{attribute addProperty BoxType ""}
{attribute addProperty Id "_defaultSyncUnitTasks_486549DC19524.3750A_0013_EL9221_4030_0018SyncUnitTasks_486549DC19524.3750A_0014_EL9221_5000_0018SyncUnitTasks_486549DC19524.3750A_0015_EL9221_5090_0018SyncUnitTasks_486549DC19524.3750A_0016_EL9221_6000_0018SyncUnitTasks_486549DC19524.3750A_0017_EL9221_6040_0018SyncUnitTasks_486549DC19524.3750A_0018_EL9221_9060_0018SyncUnitTasks_486549DC19524.3750A_0019_EL9221_9080_0018SyncUnitTasks_486549DC19524.3750A_0020_EL9222_4433_0018SyncUnitTasks_486549DC19524.3750A_0021_EL9222_5500_0018SyncUnitTasks_486549DC19524.3750A_0022_EL9222_6600_0018SyncUnitTasks_486549DC19524.3750A_0023_EL9222_6644_0018SyncUnitTasks_486549DC19524.3750A_0024_EL9222_9482_0018SyncUnitTasks_486549DC19524.3750A_0025_EL9222_9664_0018SyncUnitTasks_486549DC19524.3750A_0026_EL9227_4433_0018SyncUnitTasks_486549DC19524.3750A_0027_EL9227_5500_0018SyncUnitTasks_486549DC19524.3750A_0028_EL9227_6600_0018SyncUnitTasks_486549DC19524.3750A_0029_EL9227_6644_0018SyncUnitTasks_486549DC19524.3750A_0030_EL9227_9482_0018SyncUnitTasks_486549DC19524.3750A_0031_EL9227_9664_0018SyncUnitTasks_486549DC19524.3750A_0033_EL6690_0002_0016SyncUnitTasks_486549DC19524.3750A_0034_EL6690_0002_0017SyncUnitTasks_486549DC19524.3750A_0035_EL6690_0002_0018SyncUnitTasks_486549DC19524.3750A_0036_EL6690_0002_0019SyncUnitTasks_486549DC19524.3750A_0001_EL6720_0000_0016_0SyncUnitTasks_486549DC19524.3750A_0001_EL6720_0000_0016_1SyncUnitTasks_486549DC19524.3750A_0001_EL6720_0000_0016_2SyncUnitTasks_486549DC19524.3750A_0002_EL6720_0000_0017_0SyncUnitTasks_486549DC19524.3750A_0002_EL6720_0000_0017_1SyncUnitTasks_486549DC19524.3750A_0002_EL6720_0000_0017_2SyncUnitTasks_486549DC19524.3750A_0003_EL6720_0000_0018_0SyncUnitTasks_486549DC19524.3750A_0003_EL6720_0000_0018_1SyncUnitTasks_486549DC19524.3750A_0003_EL6720_0000_0018_2SyncUnitTasks_486549DC19524.3750A_0004_EL6720_0000_0020_0SyncUnitTasks_486549DC19524.3750A_0004_EL6720_0000_0020_1SyncUnitTasks_486549DC19524.3750A_0004_EL6720_0000_0020_2SyncUnitTasks_486549DC19524.3750A_0005_EL6731_0000_0000SyncUnitTasks_486549DC19524.3750A_0006_EL6731_0001_0000SyncUnitTasks_486549DC19524.3750A_0008_EL6731_0000_0017SyncUnitTasks_486549DC19524.3750A_0009_EL6731_0000_0018SyncUnitTasks_486549DC19524.3750A_0010_EL6731_0000_0019SyncUnitTasks_486549DC19524.3750A_0011_EL6731_0000_0020SyncUnitTasks_486549DC19524.3750A_0012_EL6731_0000_0021SyncUnitTasks_486549DC19524.3750A_0013_EL6731_0000_0022SyncUnitTasks_486549DC19524.3750A_0014_EL6731_0000_0023SyncUnitTasks_486549DC19524.3750A_0015_EL6731_0000_0025SyncUnitTasks_486549DC19524.3750A_0016_EL6731_0100_0017SyncUnitTasks_486549DC19524.3750A_0017_EL6731_0100_0018SyncUnitTasks_486549DC19524.3750A_0018_EL6731_0100_0019SyncUnitTasks_486549DC19524.3750A_0020_EL6731_0100_0021SyncUnitTasks_486549DC19524.3750A_0021_EL6731_0100_0022SyncUnitTasks_486549DC19524.3750A_0022_EL6731_0100_0023SyncUnitTasks_486549DC19524.3750A_0023_EL6731_0100_0025SyncUnitTasks_486549DC19524.3750A_0034_EL6751_0000_0000SyncUnitTasks_486549DC19524.3750A_0035_EL6751_0001_0000SyncUnitTasks_486549DC19524.3750A_0036_EL6751_0000_0016SyncUnitTasks_486549DC19524.3750A_0037_EL6751_0000_0017SyncUnitTasks_486549DC19524.3750A_0038_EL6751_0000_0018SyncUnitTasks_486549DC19524.3750A_0039_EL6751_0000_0019SyncUnitTasks_486549DC19524.3750A_0040_EL6751_0000_0021SyncUnitTasks_486549DC19524.3750A_0041_EL6751_0000_0022SyncUnitTasks_486549DC19524.3750A_0042_EL6751_0005_0022SyncUnitTasks_486549DC19524.3750A_0044_EL6751_0010_0017SyncUnitTasks_486549DC19524.3750A_0045_EL6751_0010_0018SyncUnitTasks_486549DC19524.3750A_0046_EL6751_0010_0019SyncUnitTasks_486549DC19524.3750A_0047_EL6751_0010_0021SyncUnitTasks_486549DC19524.3750A_0048_EL6752_0000_0000SyncUnitTasks_486549DC19524.3750A_0049_EL6752_0000_0016SyncUnitTasks_486549DC19524.3750A_0011_EL6861_0000_0017SyncUnitTasks_486549DC19524.3750"}
{attribute addProperty CRC "381726963"}
{attribute addProperty SizeInBites "13455"}
{attribute addProperty SizeInBytes "1681.875"}
TYPE SyncUnits_16C0B0F3 :
STRUCT
	{attribute addProperty Name "_default"}
	_default : SyncUnitTasks_486549DC;
	{attribute addProperty Name "A_0013_EL9221_4030_0018"}
	A_0013_EL9221_4030_0018 : SyncUnitTasks_486549DC;
	{attribute addProperty Name "A_0014_EL9221_5000_0018"}
	A_0014_EL9221_5000_0018 : SyncUnitTasks_486549DC;
	{attribute addProperty Name "A_0015_EL9221_5090_0018"}
	A_0015_EL9221_5090_0018 : SyncUnitTasks_486549DC;
	{attribute addProperty Name "A_0016_EL9221_6000_0018"}
	A_0016_EL9221_6000_0018 : SyncUnitTasks_486549DC;
	{attribute addProperty Name "A_0017_EL9221_6040_0018"}
	A_0017_EL9221_6040_0018 : SyncUnitTasks_486549DC;
	{attribute addProperty Name "A_0018_EL9221_9060_0018"}
	A_0018_EL9221_9060_0018 : SyncUnitTasks_486549DC;
	{attribute addProperty Name "A_0019_EL9221_9080_0018"}
	A_0019_EL9221_9080_0018 : SyncUnitTasks_486549DC;
	{attribute addProperty Name "A_0020_EL9222_4433_0018"}
	A_0020_EL9222_4433_0018 : SyncUnitTasks_486549DC;
	{attribute addProperty Name "A_0021_EL9222_5500_0018"}
	A_0021_EL9222_5500_0018 : SyncUnitTasks_486549DC;
	{attribute addProperty Name "A_0022_EL9222_6600_0018"}
	A_0022_EL9222_6600_0018 : SyncUnitTasks_486549DC;
	{attribute addProperty Name "A_0023_EL9222_6644_0018"}
	A_0023_EL9222_6644_0018 : SyncUnitTasks_486549DC;
	{attribute addProperty Name "A_0024_EL9222_9482_0018"}
	A_0024_EL9222_9482_0018 : SyncUnitTasks_486549DC;
	{attribute addProperty Name "A_0025_EL9222_9664_0018"}
	A_0025_EL9222_9664_0018 : SyncUnitTasks_486549DC;
	{attribute addProperty Name "A_0026_EL9227_4433_0018"}
	A_0026_EL9227_4433_0018 : SyncUnitTasks_486549DC;
	{attribute addProperty Name "A_0027_EL9227_5500_0018"}
	A_0027_EL9227_5500_0018 : SyncUnitTasks_486549DC;
	{attribute addProperty Name "A_0028_EL9227_6600_0018"}
	A_0028_EL9227_6600_0018 : SyncUnitTasks_486549DC;
	{attribute addProperty Name "A_0029_EL9227_6644_0018"}
	A_0029_EL9227_6644_0018 : SyncUnitTasks_486549DC;
	{attribute addProperty Name "A_0030_EL9227_9482_0018"}
	A_0030_EL9227_9482_0018 : SyncUnitTasks_486549DC;
	{attribute addProperty Name "A_0031_EL9227_9664_0018"}
	A_0031_EL9227_9664_0018 : SyncUnitTasks_486549DC;
	{attribute addProperty Name "A_0033_EL6690_0002_0016"}
	A_0033_EL6690_0002_0016 : SyncUnitTasks_486549DC;
	{attribute addProperty Name "A_0034_EL6690_0002_0017"}
	A_0034_EL6690_0002_0017 : SyncUnitTasks_486549DC;
	{attribute addProperty Name "A_0035_EL6690_0002_0018"}
	A_0035_EL6690_0002_0018 : SyncUnitTasks_486549DC;
	{attribute addProperty Name "A_0036_EL6690_0002_0019"}
	A_0036_EL6690_0002_0019 : SyncUnitTasks_486549DC;
	{attribute addProperty Name "A_0001_EL6720_0000_0016_0"}
	A_0001_EL6720_0000_0016_0 : SyncUnitTasks_486549DC;
	{attribute addProperty Name "A_0001_EL6720_0000_0016_1"}
	A_0001_EL6720_0000_0016_1 : SyncUnitTasks_486549DC;
	{attribute addProperty Name "A_0001_EL6720_0000_0016_2"}
	A_0001_EL6720_0000_0016_2 : SyncUnitTasks_486549DC;
	{attribute addProperty Name "A_0002_EL6720_0000_0017_0"}
	A_0002_EL6720_0000_0017_0 : SyncUnitTasks_486549DC;
	{attribute addProperty Name "A_0002_EL6720_0000_0017_1"}
	A_0002_EL6720_0000_0017_1 : SyncUnitTasks_486549DC;
	{attribute addProperty Name "A_0002_EL6720_0000_0017_2"}
	A_0002_EL6720_0000_0017_2 : SyncUnitTasks_486549DC;
	{attribute addProperty Name "A_0003_EL6720_0000_0018_0"}
	A_0003_EL6720_0000_0018_0 : SyncUnitTasks_486549DC;
	{attribute addProperty Name "A_0003_EL6720_0000_0018_1"}
	A_0003_EL6720_0000_0018_1 : SyncUnitTasks_486549DC;
	{attribute addProperty Name "A_0003_EL6720_0000_0018_2"}
	A_0003_EL6720_0000_0018_2 : SyncUnitTasks_486549DC;
	{attribute addProperty Name "A_0004_EL6720_0000_0020_0"}
	A_0004_EL6720_0000_0020_0 : SyncUnitTasks_486549DC;
	{attribute addProperty Name "A_0004_EL6720_0000_0020_1"}
	A_0004_EL6720_0000_0020_1 : SyncUnitTasks_486549DC;
	{attribute addProperty Name "A_0004_EL6720_0000_0020_2"}
	A_0004_EL6720_0000_0020_2 : SyncUnitTasks_486549DC;
	{attribute addProperty Name "A_0005_EL6731_0000_0000"}
	A_0005_EL6731_0000_0000 : SyncUnitTasks_486549DC;
	{attribute addProperty Name "A_0006_EL6731_0001_0000"}
	A_0006_EL6731_0001_0000 : SyncUnitTasks_486549DC;
	{attribute addProperty Name "A_0008_EL6731_0000_0017"}
	A_0008_EL6731_0000_0017 : SyncUnitTasks_486549DC;
	{attribute addProperty Name "A_0009_EL6731_0000_0018"}
	A_0009_EL6731_0000_0018 : SyncUnitTasks_486549DC;
	{attribute addProperty Name "A_0010_EL6731_0000_0019"}
	A_0010_EL6731_0000_0019 : SyncUnitTasks_486549DC;
	{attribute addProperty Name "A_0011_EL6731_0000_0020"}
	A_0011_EL6731_0000_0020 : SyncUnitTasks_486549DC;
	{attribute addProperty Name "A_0012_EL6731_0000_0021"}
	A_0012_EL6731_0000_0021 : SyncUnitTasks_486549DC;
	{attribute addProperty Name "A_0013_EL6731_0000_0022"}
	A_0013_EL6731_0000_0022 : SyncUnitTasks_486549DC;
	{attribute addProperty Name "A_0014_EL6731_0000_0023"}
	A_0014_EL6731_0000_0023 : SyncUnitTasks_486549DC;
	{attribute addProperty Name "A_0015_EL6731_0000_0025"}
	A_0015_EL6731_0000_0025 : SyncUnitTasks_486549DC;
	{attribute addProperty Name "A_0016_EL6731_0100_0017"}
	A_0016_EL6731_0100_0017 : SyncUnitTasks_486549DC;
	{attribute addProperty Name "A_0017_EL6731_0100_0018"}
	A_0017_EL6731_0100_0018 : SyncUnitTasks_486549DC;
	{attribute addProperty Name "A_0018_EL6731_0100_0019"}
	A_0018_EL6731_0100_0019 : SyncUnitTasks_486549DC;
	{attribute addProperty Name "A_0020_EL6731_0100_0021"}
	A_0020_EL6731_0100_0021 : SyncUnitTasks_486549DC;
	{attribute addProperty Name "A_0021_EL6731_0100_0022"}
	A_0021_EL6731_0100_0022 : SyncUnitTasks_486549DC;
	{attribute addProperty Name "A_0022_EL6731_0100_0023"}
	A_0022_EL6731_0100_0023 : SyncUnitTasks_486549DC;
	{attribute addProperty Name "A_0023_EL6731_0100_0025"}
	A_0023_EL6731_0100_0025 : SyncUnitTasks_486549DC;
	{attribute addProperty Name "A_0034_EL6751_0000_0000"}
	A_0034_EL6751_0000_0000 : SyncUnitTasks_486549DC;
	{attribute addProperty Name "A_0035_EL6751_0001_0000"}
	A_0035_EL6751_0001_0000 : SyncUnitTasks_486549DC;
	{attribute addProperty Name "A_0036_EL6751_0000_0016"}
	A_0036_EL6751_0000_0016 : SyncUnitTasks_486549DC;
	{attribute addProperty Name "A_0037_EL6751_0000_0017"}
	A_0037_EL6751_0000_0017 : SyncUnitTasks_486549DC;
	{attribute addProperty Name "A_0038_EL6751_0000_0018"}
	A_0038_EL6751_0000_0018 : SyncUnitTasks_486549DC;
	{attribute addProperty Name "A_0039_EL6751_0000_0019"}
	A_0039_EL6751_0000_0019 : SyncUnitTasks_486549DC;
	{attribute addProperty Name "A_0040_EL6751_0000_0021"}
	A_0040_EL6751_0000_0021 : SyncUnitTasks_486549DC;
	{attribute addProperty Name "A_0041_EL6751_0000_0022"}
	A_0041_EL6751_0000_0022 : SyncUnitTasks_486549DC;
	{attribute addProperty Name "A_0042_EL6751_0005_0022"}
	A_0042_EL6751_0005_0022 : SyncUnitTasks_486549DC;
	{attribute addProperty Name "A_0044_EL6751_0010_0017"}
	A_0044_EL6751_0010_0017 : SyncUnitTasks_486549DC;
	{attribute addProperty Name "A_0045_EL6751_0010_0018"}
	A_0045_EL6751_0010_0018 : SyncUnitTasks_486549DC;
	{attribute addProperty Name "A_0046_EL6751_0010_0019"}
	A_0046_EL6751_0010_0019 : SyncUnitTasks_486549DC;
	{attribute addProperty Name "A_0047_EL6751_0010_0021"}
	A_0047_EL6751_0010_0021 : SyncUnitTasks_486549DC;
	{attribute addProperty Name "A_0048_EL6752_0000_0000"}
	A_0048_EL6752_0000_0000 : SyncUnitTasks_486549DC;
	{attribute addProperty Name "A_0049_EL6752_0000_0016"}
	A_0049_EL6752_0000_0016 : SyncUnitTasks_486549DC;
	{attribute addProperty Name "A_0011_EL6861_0000_0017"}
	A_0011_EL6861_0000_0017 : SyncUnitTasks_486549DC;
END_STRUCT
END_TYPE

(* stored: Version 1.2.0.0, ProductVersion 3.1.4024.9
   DUT SyncUnits_16C0B0F3: Id {4213f188-ff11-4ba1-be1b-a4d13e115dc7} *)
